// TIA Portal V18 export
// export: Created 2026-04-18T00:00:00Z, ExportSetting WithDefaults
FUNCTION_BLOCK "FB_Tu_Dong"   // FB100, LAD
{ S7_Optimized_Access := 'TRUE' }
VERSION : 0.1
// stored: AutoNumber true, IsIECCheckEnabled false, IsRetainMemResEnabled false
   VAR
      Timer_Van : IEC_TIMER;
   END_VAR
BEGIN

REGION Network 1: Khởi động động cơ
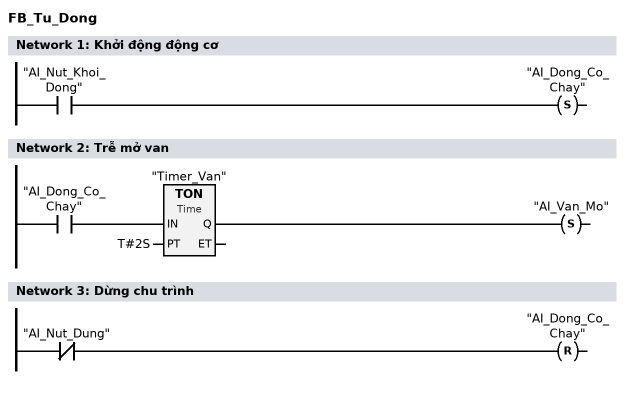
   RUNG wire#powerrail
      Contact( "AI_Nut_Khoi_Dong" )
      S_Coil( "AI_Dong_Co_Chay" )
   END_RUNG
   // the same network as SCL:
   IF "AI_Nut_Khoi_Dong" THEN "AI_Dong_Co_Chay" := TRUE; END_IF;
END_REGION

REGION Network 2: Trễ mở van
   RUNG wire#powerrail
      Contact( "AI_Dong_Co_Chay" )
      { S7_Templates := "time_type := Time" } "Timer_Van".TON(pt := T#2S, et =>)
      S_Coil( "AI_Van_Mo" )
   END_RUNG
   // the same network as SCL:
   "Timer_Van".TON(IN := "AI_Dong_Co_Chay", PT := T#2S);
   IF "Timer_Van".Q THEN "AI_Van_Mo" := TRUE; END_IF;
END_REGION

REGION Network 3: Dừng chu trình
   RUNG wire#powerrail
      I_Contact( "AI_Nut_Dung" )
      R_Coil( "AI_Dong_Co_Chay" )
   END_RUNG
   // the same network as SCL:
   IF NOT "AI_Nut_Dung" THEN "AI_Dong_Co_Chay" := FALSE; END_IF;
END_REGION
END_FUNCTION_BLOCK
